FUNCTION_BLOCK ConvertFlowUnit (* Basic Function Block Type *)
  (* Standard: 61499-2 *)
  (* Version 0.0, 8/23/2024, SESA713705, Schneider Electric, Template *)
  PACKAGE SE.Nereda;
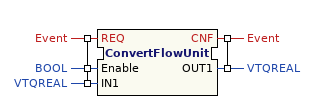
  EVENT_INPUT
    REQ WITH IN1, Enable; (* Normal Execution Request *)
  END_EVENT
  EVENT_OUTPUT
    CNF WITH OUT1; (* Execution Confirmation *)
  END_EVENT
  VAR_INPUT
    Enable : BOOL;
    IN1 : VTQREAL; (* Input event qualifier *)
  END_VAR
  VAR_OUTPUT
    OUT1 : VTQREAL; (* Output event qualifier *)
  END_VAR
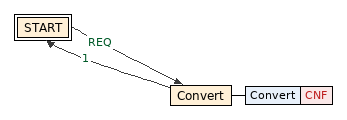
  EC_STATES
    START; (* Initial State *)
    Convert : Convert -> CNF;
  END_STATES
  EC_TRANSITIONS
    START TO Convert := REQ;
    Convert TO START := 1;
  END_TRANSITIONS
  ALGORITHM Convert IN ST:
;
IF Enable THEN
	// flow conversion from m3/s to m3/h
	OUT1.value := IN1.value * 3.6;
	OUT1.timestamp := IN1.timestamp;
	OUT1.picosecs := IN1.picosecs;
	OUT1.quality := IN1.quality;
ELSE
	OUT1 := IN1;
END_IF;
  END_ALGORITHM
END_FUNCTION_BLOCK
